FUNCTION FN_StringToLane : cLaneSel
VAR_INPUT
	Lane: STRING(30);
END_VAR

//Determin lane from string input
IF Lane = TO_STRING(cLaneSel.Green) THEN
	FN_StringToLane := cLaneSel.Green;
ELSIF Lane = TO_STRING(cLaneSel.Red) THEN
	FN_StringToLane := cLaneSel.Red;
ELSIF Lane = TO_STRING(cLaneSel.Blue) THEN
	FN_StringToLane := cLaneSel.Blue;
ELSE
	FN_StringToLane := cLaneSel.None;
END_IF

END_FUNCTION

(* stored: Version 1.1.0.1, ProductVersion 3.1.4024.6
   POU FN_StringToLane: Id {ad787d43-1891-410e-aa38-653843f1c4cc}, SpecialFunc None *)
